Yaskawa INFORM job: R1_72,2(0,0)R2.JBI

/JOB
//NAME R1_72,2(0,0)R2
///FOLDERNAME KRIS-SCIANA
//POS
///NPOS 51,51,0,3,0,0
///TOOL 0
///POSTYPE PULSE
///PULSE
C00000=-120731,-9924,-70355,-68051,94259,-38782
C00001=-120731,-9924,-44892,-68051,94259,-38782
C00002=-120731,-9924,-44892,-68051,94259,-38782
C00003=-127639,-20983,-36057,-64456,72146,-38182
C00004=-128458,-18258,-30093,-64911,70598,-37327
C00005=-128458,-18212,-29006,-65109,70310,-37046
C00006=-128458,-18258,-30093,-64911,70598,-37327
C00007=-129158,-18100,-29977,-64744,70152,-37441
C00008=-128458,-18258,-30093,-64911,70598,-37327
C00009=-120732,-29819,-84626,-67909,93683,-38165
C00010=-120732,-29819,-84626,-67909,93683,-38165
C00011=-116404,-32627,-69232,-81055,84641,-52345
C00012=-125149,-29195,-64737,-78117,78810,-52454
C00013=-126167,-29055,-64642,-77752,78161,-52536
C00014=-125149,-29195,-64737,-78117,78810,-52454
C00015=-125149,-27912,-66309,-77844,79197,-53197
C00016=-130097,-20035,-71206,-66140,83686,-56378
C00017=-130097,-20918,-70680,-66200,83352,-56048
C00018=-130097,-20035,-71206,-66140,83686,-56378
C00019=-135693,-32727,-79902,-63722,80117,-56600
C00020=-162052,-74362,-107056,-19862,52172,-63712
C00021=-160626,-67164,-100928,-21065,52420,-63197
C00022=-160165,-65351,-100040,-21338,52886,-63117
C00023=-160626,-67164,-100928,-21065,52420,-63197
C00024=-163319,-77470,-105726,-19436,49622,-63701
C00025=-159440,-68974,-103163,-21917,53108,-62878
C00026=-158867,-65638,-101075,-22266,53641,-62772
C00027=-118936,-86323,-121653,-1041,96543,53661
///LIMIT ON
C00028=-120737,-316086,375860,-1155,25196,53627
///LIMIT OFF
C00029=-159355,-64693,-100608,-21817,53712,-62976
C00030=-162669,-60415,-98452,-18893,53815,-64266
C00031=-186148,-6414,-82548,19704,93724,-60581
C00032=-186030,-5612,-81909,19644,93725,-60553
C00033=-175537,27291,-64588,6081,111496,-60595
C00034=-177455,28166,-68259,7068,114275,-60836
C00035=-143288,-43790,-101806,-35807,79991,-60997
C00036=-144672,-29256,-89797,-35009,79619,-61314
///LIMIT ON
C00037=38711,-128331,-123199,-49626,97531,112150
C00038=37108,-130734,-125310,-49549,96709,111766
///LIMIT OFF
C00039=-144373,-16278,-85433,-34732,88432,-64092
C00040=-145220,-22654,-89314,-34279,87450,-64033
C00041=-145391,-24453,-90442,-34190,87209,-64008
C00042=-147427,-52289,-112602,-33103,86067,-64259
C00043=-120731,-9924,-70355,-68051,94259,-38782
C00044=-124666,-10874,-42026,-56973,84332,-28663
C00045=-127583,-8457,-31565,-56644,79715,-27199
C00046=-128641,-4479,-26552,-56509,78511,-26996
C00047=-128167,3287,-20176,-56623,78825,-26931
C00048=-127452,-4898,-29666,-56592,80169,-27427
C00049=-115096,-48686,-81785,-59858,92460,-29001
C00050=-2836,-82790,-98931,5475,98593,-23263
BC00000=248830,665841,1065590
BC00001=248830,665841,393906
BC00002=254751,691106,393906
BC00003=254751,691106,393906
BC00004=254751,691106,393906
BC00005=254751,691106,393906
BC00006=254751,691106,393906
BC00007=254751,691106,393906
BC00008=254751,691106,393906
BC00009=248830,678392,941452
BC00010=265899,731832,938155
BC00011=265899,731832,938155
BC00012=257495,731832,938155
BC00013=257495,731832,938155
BC00014=257495,731832,938155
BC00015=257495,731832,938155
BC00016=257495,731832,938155
BC00017=257495,731832,938155
BC00018=257495,731832,938155
BC00019=257495,731832,938155
BC00020=257495,731832,938155
BC00021=257495,731832,938155
BC00022=257495,731832,938155
BC00023=257495,731832,938155
BC00024=257495,731832,938155
BC00025=257495,731832,938155
BC00026=257495,731832,938155
///LIMIT ON
BC00027=145924,651668,1070910
BC00028=145924,651668,1070910
///LIMIT OFF
BC00029=257495,731832,938155
BC00030=257495,731832,938155
BC00031=257495,731832,938155
BC00032=257495,731832,938155
BC00033=257495,731832,938155
BC00034=257495,731832,938155
BC00035=257495,731832,938155
BC00036=257495,731832,938155
BC00037=17998,679451,1070910
BC00038=17998,679451,1070910
BC00039=257495,731832,938155
BC00040=257495,731832,938155
BC00041=257495,731832,938155
BC00042=257495,731832,938155
BC00043=248830,665841,1065590
BC00044=248830,677088,383396
BC00045=248830,677088,383396
BC00046=248830,677088,383396
BC00047=248830,677088,383396
BC00048=248830,677088,383396
BC00049=248830,677088,383396
BC00050=102451,677088,953097
///POSTYPE BASE
///RECTAN
///RCONF 0,0,0,0,0,0,0,0,0,0,0,0,0,0,0,0,0,0,0,0,0,0,0,0
P00006=0.222,-3.123,-1.508,0.0000,0.0000,0.0000
P00021=-0.225,-6.128,-0.405,0.0000,0.0000,0.0000
P00030=5.926,-4.294,-1.390,0.0000,0.0000,0.0000
//INST
///DATE 2024/07/24 14:07
///ATTR SC,RW
///GROUP1 RB1,BS1
NOP
'R2_72.2(0,0)
'Path S1184
SFTOF
MOVJ C00000 BC00000 VJ=100.00
MOVJ C00001 BC00001 VJ=100.00
MOVJ C00002 BC00002 VJ=100.00
MOVL C00003 BC00003 V=333.3
MOVL C00004 BC00004 V=100.0
REFP 3 C00005 BC00005
CALL JOB:SEARCH-R1
SET P030 P006
SFTON P030
MOVL C00006 BC00006 V=100.0
REFP 3 C00007 BC00007
CALL JOB:SEARCH-R1
SET P030 P006
SFTON P030
MOVL C00008 BC00008 V=100.0
SFTOF
MOVJ C00009 BC00009 VJ=100.00
MOVJ C00010 BC00010 VJ=100.00
MOVL C00011 BC00011 V=333.3
MOVL C00012 BC00012 V=100.0
REFP 3 C00013 BC00013
CALL JOB:SEARCH-R1
SET P021 P006
SFTON P021
MOVL C00014 BC00014 V=250.0
MOVL C00015 BC00015 V=250.0
MOVL C00016 BC00016 V=166.7
REFP 3 C00017 BC00017
CALL JOB:SEARCH-R1
SET P021 P006
SFTON P021
MOVL C00018 BC00018 V=166.7
MOVL C00019 BC00019 V=333.3
MOVL C00020 BC00020 V=333.3
MOVL C00021 BC00021 V=166.7
REFP 3 C00022 BC00022
CALL JOB:SEARCH-R1
SET P021 P006
SFTON P021
MOVL C00023 BC00023 V=166.7
SFTOF
MOVL C00024 BC00024 V=166.7
MOVL C00025 BC00025 V=166.7
'Path W1186
SFTOF
SFTON P021
MOVL C00026 BC00026 V=100.0 PL=0
REFP 1 C00027 BC00027
REFP 2 C00028 BC00028
MACRO1 MJ#(0) ARGF6
ARCON
MOVL C00029 BC00029 V=10.8
MOVL C00030 BC00030 V=10.8
ARCOF
MOVL C00031 BC00031 V=10.0
ARCON
MOVL C00032 BC00032 V=11.7
MOVL C00033 BC00033 V=12.3
ARCOF
MOVL C00034 BC00034 V=250.0
MOVL C00035 BC00035 V=333.3
SFTOF
'Path W1188
SFTOF
SFTON P021
MOVL C00036 BC00036 V=250.0 PL=0
REFP 1 C00037 BC00037
REFP 2 C00038 BC00038
MACRO1 MJ#(0) ARGF6
ARCON
MOVL C00039 BC00039 V=8.3
MOVL C00040 BC00040 V=8.3
MOVL C00041 BC00041 V=8.3
ARCOF
MOVL C00042 BC00042 V=333.3
SFTOF
MOVJ C00043 BC00043 VJ=100.00
MOVL C00044 BC00044 V=833.3
SFTON P030
MOVL C00045 BC00045 V=166.7
MOVL C00046 BC00046 V=166.7 PL=0
MACRO1 MJ#(0) ARGF7
ARCON
MOVL C00047 BC00047 V=9.2
ARCOF
MOVL C00048 BC00048 V=166.7
SFTOF
MOVJ C00049 BC00049 VJ=100.00
MOVJ C00050 BC00050 VJ=100.00
SFTOF
END
